{attribute addProperty BoxType "EK1122-0000-0018"}
{attribute addProperty Id "Beckhoff_AX88xxsub_EK1100EK1100_179A0949162"}
{attribute addProperty CRC "669120792"}
{attribute addProperty SizeInBites "16"}
{attribute addProperty SizeInBytes "2"}
TYPE Beckhoff_AX88xxEK1122_27E1F918 EXTENDS EK1122_179A0949 :
STRUCT
	{attribute addProperty Name "Beckhoff_AX88xxsub_EK1100"}
	Beckhoff_AX88xxsub_EK1100 : EK1100_179A0949;
END_STRUCT
END_TYPE

(* stored: Version 1.2.0.0, ProductVersion 3.1.4024.9
   DUT Beckhoff_AX88xxEK1122_27E1F918: Id {0e551f70-d57a-4ca5-80fc-9736711be6a0} *)
